SYSTEM VAV_MVCL (* Variable Air Valve System Model+View+Control+HMI *)
  (* Standard: IEC 61499-1; Classification: Simulation; ApplicationDomain: HVAC *)
  (* Version 0.0, 2006-04-27, JHC, Holobloc Inc, Derived from VAV_MVL. *)
  DEVICE HMI : FRAME_DEVICE(BOUNDS := [100,100,140,270])
    RESOURCE FP : PANEL_RESOURCE (* Controller Faceplate *)
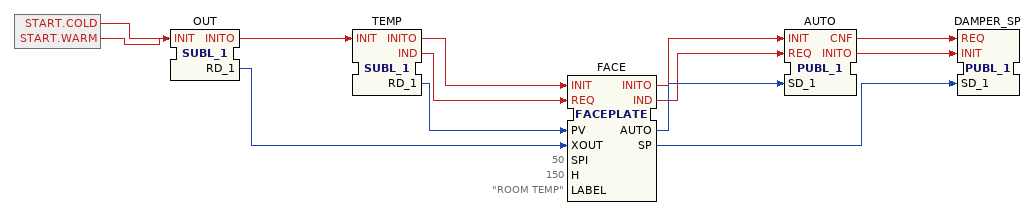
      FBS
        TEMP : SUBL_1;
        FACE : FACEPLATE(SPI := 50, H := 150, LABEL := "ROOM TEMP");
        OUT : SUBL_1;
        AUTO : PUBL_1;
        DAMPER_SP : PUBL_1;
      END_FBS
      EVENT_CONNECTIONS
        FACE.INITO TO AUTO.INIT;
        FACE.IND TO AUTO.REQ;
        START.COLD TO OUT.INIT;
        START.WARM TO OUT.INIT;
        OUT.INITO TO TEMP.INIT;
        TEMP.INITO TO FACE.INIT;
        TEMP.IND TO FACE.REQ;
        AUTO.CNF TO DAMPER_SP.REQ;
        AUTO.INITO TO DAMPER_SP.INIT;
      END_CONNECTIONS
      DATA_CONNECTIONS
        TEMP.RD_1 TO FACE.PV;
        OUT.RD_1 TO FACE.XOUT;
        FACE.AUTO TO AUTO.SD_1;
        FACE.SP TO DAMPER_SP.SD_1;
      END_CONNECTIONS
    END_RESOURCE
  END_DEVICE
  DEVICE RECORDER : FRAME_DEVICE(BOUNDS := [240,100,210,250])
    RESOURCE RECORDER : PANEL_RESOURCE
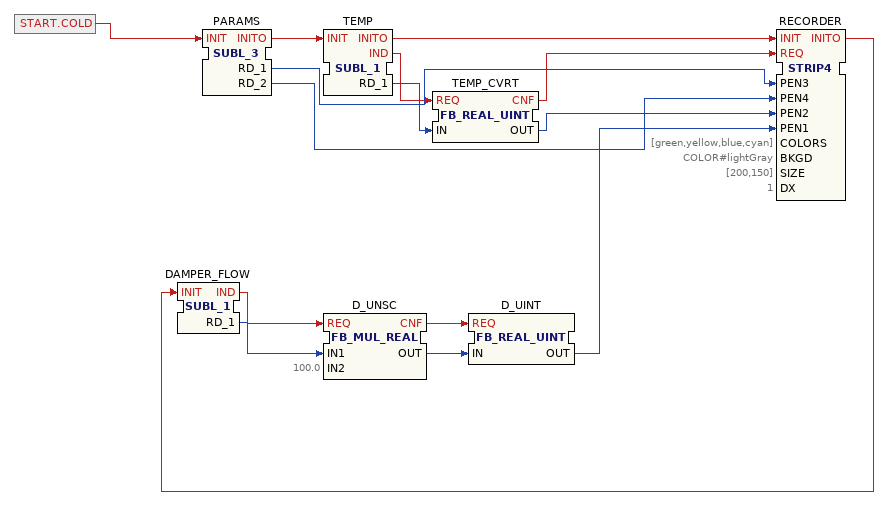
      FBS
        RECORDER : STRIP4(COLORS := [green,yellow,blue,cyan], BKGD := COLOR#lightGray, SIZE := [200,150], DX := 1);
        TEMP : SUBL_1;
        PARAMS : SUBL_3;
        DAMPER_FLOW : SUBL_1;
        TEMP_CVRT : FB_REAL_UINT;
        D_UNSC : FB_MUL_REAL(IN2 := 100.0);
        D_UINT : FB_REAL_UINT;
      END_FBS
      EVENT_CONNECTIONS
        START.COLD TO PARAMS.INIT;
        TEMP.INITO TO RECORDER.INIT;
        TEMP.IND TO TEMP_CVRT.REQ;
        TEMP_CVRT.CNF TO RECORDER.REQ;
        PARAMS.INITO TO TEMP.INIT;
        RECORDER.INITO TO DAMPER_FLOW.INIT;
        D_UNSC.CNF TO D_UINT.REQ;
        DAMPER_FLOW.IND TO D_UNSC.REQ;
      END_CONNECTIONS
      DATA_CONNECTIONS
        PARAMS.RD_1 TO RECORDER.PEN3;
        PARAMS.RD_2 TO RECORDER.PEN4;
        TEMP.RD_1 TO TEMP_CVRT.IN;
        TEMP_CVRT.OUT TO RECORDER.PEN2;
        D_UNSC.OUT TO D_UINT.IN;
        D_UINT.OUT TO RECORDER.PEN1;
        DAMPER_FLOW.RD_1 TO D_UNSC.IN1;
      END_CONNECTIONS
    END_RESOURCE
    RESOURCE PARAMS : PANEL_RESOURCE(ROWS := 2, COLS := 2)
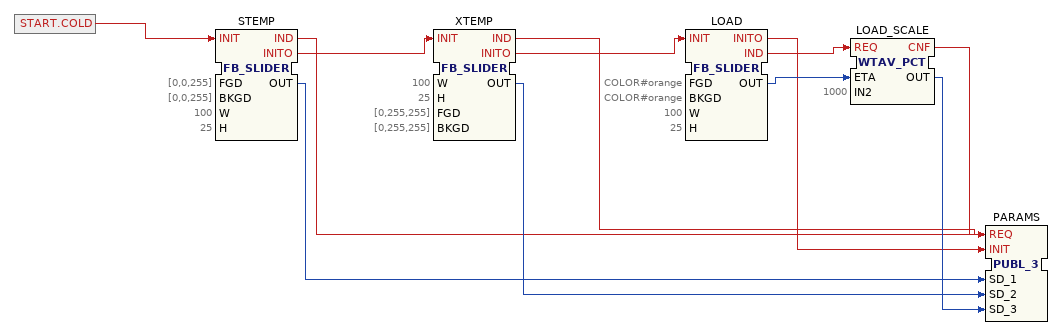
      FBS
        PARAMS : PUBL_3;
        STEMP : FB_SLIDER(FGD := [0,0,255], BKGD := [0,0,255], W := 100, H := 25);
        XTEMP : FB_SLIDER(W := 100, H := 25, FGD := [0,255,255], BKGD := [0,255,255]);
        LOAD : FB_SLIDER(FGD := COLOR#orange, BKGD := COLOR#orange, W := 100, H := 25);
        LOAD_SCALE : WTAV_PCT(IN2 := 1000);
      END_FBS
      EVENT_CONNECTIONS
        STEMP.IND TO PARAMS.REQ;
        STEMP.INITO TO XTEMP.INIT;
        XTEMP.IND TO PARAMS.REQ;
        XTEMP.INITO TO LOAD.INIT;
        LOAD.INITO TO PARAMS.INIT;
        START.COLD TO STEMP.INIT;
        LOAD.IND TO LOAD_SCALE.REQ;
        LOAD_SCALE.CNF TO PARAMS.REQ;
      END_CONNECTIONS
      DATA_CONNECTIONS
        STEMP.OUT TO PARAMS.SD_1;
        XTEMP.OUT TO PARAMS.SD_2;
        LOAD.OUT TO LOAD_SCALE.ETA;
        LOAD_SCALE.OUT TO PARAMS.SD_3;
      END_CONNECTIONS
    END_RESOURCE
  END_DEVICE
  DEVICE MV : FRAME_DEVICE(BOUNDS := [450,100,290,250]) (* Room/Duct Model + View *)
    RESOURCE MODEL : EMB_RES
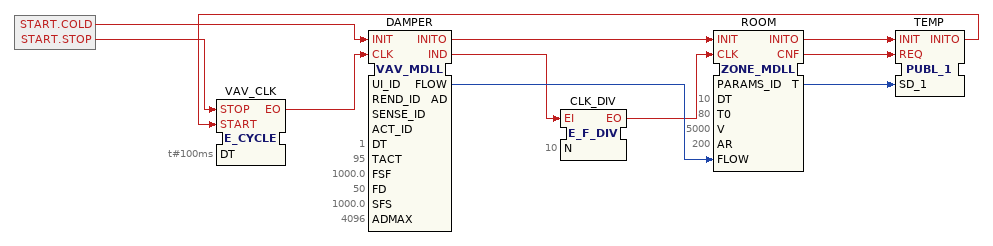
      FBS
        DAMPER : VAV_MDLL(DT := 1, TACT := 95, FSF := 1000.0, FD := 50, SFS := 1000.0, ADMAX := 4096);
        ROOM : ZONE_MDLL(DT := 10, T0 := 80, V := 5000, AR := 200);
        CLK_DIV : E_F_DIV(N := 10); (* Zone simulation runs 10x slower than valve sim *)
        VAV_CLK : E_CYCLE(DT := t#100ms);
        TEMP : PUBL_1; (* Main Display clock and Temperature publisher *)
      END_FBS
      EVENT_CONNECTIONS
        START.COLD TO DAMPER.INIT;
        DAMPER.INITO TO ROOM.INIT;
        DAMPER.IND TO CLK_DIV.EI;
        CLK_DIV.EO TO ROOM.CLK;
        START.STOP TO VAV_CLK.STOP;
        VAV_CLK.EO TO DAMPER.CLK;
        ROOM.INITO TO TEMP.INIT;
        TEMP.INITO TO VAV_CLK.START;
        ROOM.CNF TO TEMP.REQ;
      END_CONNECTIONS
      DATA_CONNECTIONS
        DAMPER.FLOW TO ROOM.FLOW;
        ROOM.T TO TEMP.SD_1;
      END_CONNECTIONS
    END_RESOURCE
    RESOURCE DUCTS : VIEW_PANEL(DIA := 25, SIZE := [3,8], VERTICAL := 1)
      FBS
        DAMPER : MECH_VIEW(BKGD := [0,0,255], DIR := 0, STYLE := VSTYLE#DAMPER, WKPC := [0,255,0], LEN := 3);
        LBLS : XSPACE(LBLS := ["","===>","","",""], DIMS := [3,6], COLORS := [green,white]);
        OUTLET : XSPACE(COLORS := [yellow,blue], DIMS := [3,1], LBLS := ["","","","","<==="]);
        DAMPER_UI : PUBL_1;
        DAMPER_REND : SUBL_1;
      END_FBS
      EVENT_CONNECTIONS
        LBLS.INITO TO OUTLET.INIT;
        DAMPER.INITO TO DAMPER_UI.INIT;
        DAMPER.IND TO DAMPER_UI.REQ;
        DAMPER_UI.INITO TO LBLS.INIT;
        START.COLD TO DAMPER_REND.INIT;
        DAMPER_REND.INITO TO DAMPER.INIT;
        DAMPER_REND.IND TO DAMPER.REQ;
      END_CONNECTIONS
      DATA_CONNECTIONS
        DAMPER.FAULT TO DAMPER_UI.SD_1;
        DAMPER_REND.RD_1 TO DAMPER.POS;
      END_CONNECTIONS
    END_RESOURCE
    RESOURCE ROOM : VIEW_PANEL(SIZE := [8,8], DIA := 25)
      FBS
        ROOM : ZONE_VIEWL(FGD := [255,255,0], BKGD := [0,0,255], W := 200, SZ := 14, REND_ID := "DAMPER_REND");
        TEMP : SUBL_1;
      END_FBS
      EVENT_CONNECTIONS
        START.COLD TO TEMP.INIT;
        START.WARM TO TEMP.INIT;
        TEMP.INITO TO ROOM.INIT;
        TEMP.IND TO ROOM.REQ;
      END_CONNECTIONS
      DATA_CONNECTIONS
        TEMP.RD_1 TO ROOM.TEMP;
      END_CONNECTIONS
    END_RESOURCE
  END_DEVICE
  DEVICE DAMPER : FRAME_DEVICE(BOUNDS := [240,350,160,170], GRID := [1,1])
    RESOURCE HMI : PANEL_RESOURCE
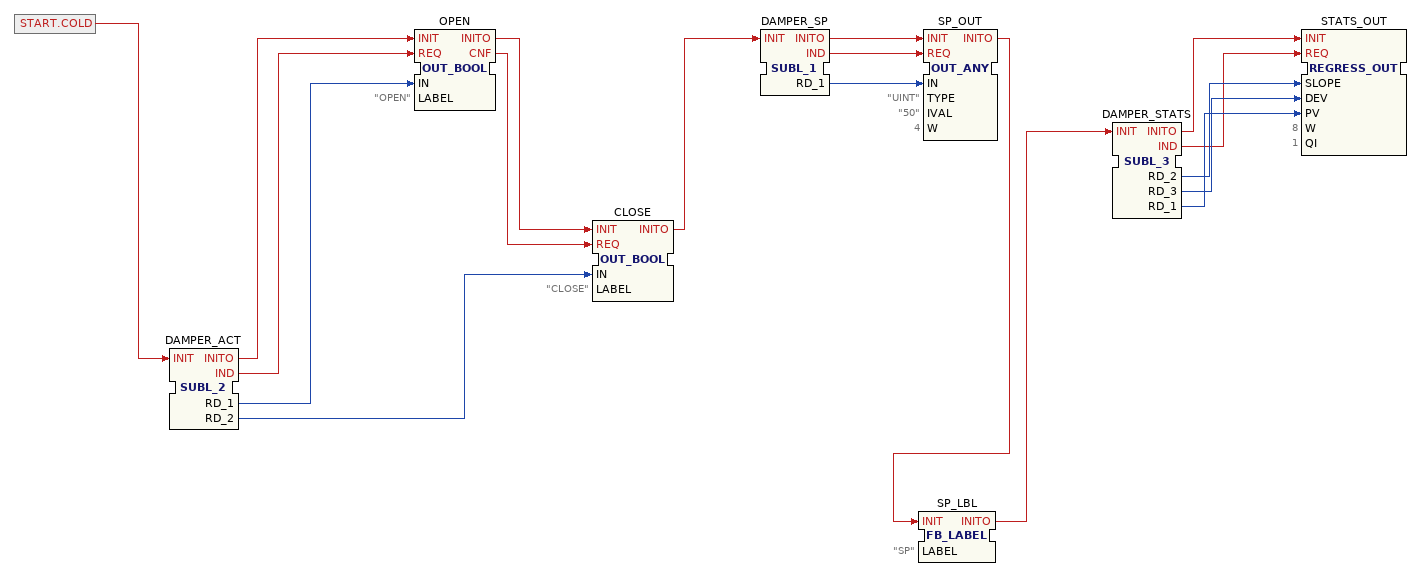
      FBS
        DAMPER_ACT : SUBL_2;
        DAMPER_SP : SUBL_1;
        SP_OUT : OUT_ANY(TYPE := "UINT", IVAL := "50", W := 4);
        SP_LBL : FB_LABEL(LABEL := "SP");
        DAMPER_STATS : SUBL_3;
        OPEN : OUT_BOOL(LABEL := "OPEN");
        CLOSE : OUT_BOOL(LABEL := "CLOSE");
        STATS_OUT : REGRESS_OUT(W := 8, QI := 1);
      END_FBS
      EVENT_CONNECTIONS
        DAMPER_SP.INITO TO SP_OUT.INIT;
        DAMPER_SP.IND TO SP_OUT.REQ;
        SP_OUT.INITO TO SP_LBL.INIT;
        SP_LBL.INITO TO DAMPER_STATS.INIT;
        START.COLD TO DAMPER_ACT.INIT;
        DAMPER_ACT.INITO TO OPEN.INIT;
        DAMPER_ACT.IND TO OPEN.REQ;
        OPEN.INITO TO CLOSE.INIT;
        OPEN.CNF TO CLOSE.REQ;
        CLOSE.INITO TO DAMPER_SP.INIT;
        DAMPER_STATS.INITO TO STATS_OUT.INIT;
        DAMPER_STATS.IND TO STATS_OUT.REQ;
      END_CONNECTIONS
      DATA_CONNECTIONS
        DAMPER_SP.RD_1 TO SP_OUT.IN;
        DAMPER_ACT.RD_1 TO OPEN.IN;
        DAMPER_ACT.RD_2 TO CLOSE.IN;
        DAMPER_STATS.RD_2 TO STATS_OUT.SLOPE;
        DAMPER_STATS.RD_3 TO STATS_OUT.DEV;
        DAMPER_STATS.RD_1 TO STATS_OUT.PV;
      END_CONNECTIONS
    END_RESOURCE
    RESOURCE CTRL : EMB_RES
      FBS
        DAMPER_SENSE : SUBL_1; (* A/D Reading *)
        DIV : E_F_DIV(N := 10); (* Display every 10 A/D cycles *)
        SCALER : SCALE_UR(MAX := 4096);
        STATS : REGRESS(N := 10);
        DAMPER_FLOW : PUBL_1;
        FLOW_CVRT : FB_SQRT; (* Convert delta-P to flow units *)
        DAMPER_STATS : PUBL_3;
        DCTL : DAMPER_CTL;
        DAMPER_ACT : PUBL_2;
        DAMPER_SP : SUBL_1;
        SP_CVRT : FB_UINT_REAL;
        SP_SCALE : FB_MUL_REAL(IN2 := 0.01);
      END_FBS
      EVENT_CONNECTIONS
        START.COLD TO DAMPER_SENSE.INIT;
        START.WARM TO DAMPER_SENSE.INIT;
        DAMPER_SENSE.IND TO SCALER.REQ;
        DAMPER_SENSE.INITO TO STATS.INIT;
        STATS.CNF TO DIV.EI;
        DAMPER_FLOW.INITO TO DIV.R;
        SCALER.CNF TO FLOW_CVRT.REQ;
        FLOW_CVRT.CNF TO DAMPER_FLOW.REQ;
        DAMPER_FLOW.CNF TO STATS.REQ;
        STATS.INITO TO DAMPER_STATS.INIT;
        DIV.EO TO DAMPER_STATS.REQ;
        DAMPER_STATS.CNF TO DCTL.REQ;
        DAMPER_STATS.INITO TO DCTL.INIT;
        DCTL.INITO TO DAMPER_ACT.INIT;
        DCTL.CNF TO DAMPER_ACT.REQ;
        DAMPER_ACT.INITO TO DAMPER_SP.INIT;
        DAMPER_SP.IND TO SP_CVRT.REQ;
        SP_CVRT.CNF TO SP_SCALE.REQ;
        DAMPER_SP.INITO TO DAMPER_FLOW.INIT;
      END_CONNECTIONS
      DATA_CONNECTIONS
        DAMPER_SENSE.RD_1 TO SCALER.IN;
        FLOW_CVRT.OUT TO DAMPER_FLOW.SD_1;
        SCALER.OUT TO FLOW_CVRT.IN;
        FLOW_CVRT.OUT TO STATS.IN;
        STATS.OUT TO DAMPER_STATS.SD_1;
        STATS.SLOPE TO DAMPER_STATS.SD_2;
        STATS.DEV TO DAMPER_STATS.SD_3;
        STATS.OUT TO DCTL.PV;
        STATS.SLOPE TO DCTL.SLOPE;
        STATS.DEV TO DCTL.DEV;
        DCTL.OPEN TO DAMPER_ACT.SD_1;
        DCTL.CLOSE TO DAMPER_ACT.SD_2;
        DAMPER_SP.RD_1 TO SP_CVRT.IN;
        SP_CVRT.OUT TO SP_SCALE.IN1;
        SP_SCALE.OUT TO DCTL.SP;
      END_CONNECTIONS
    END_RESOURCE
  END_DEVICE
END_SYSTEM
